// TIA Portal V15.1 export
// export: Created 2022-12-20T09:13:23.4021244Z, ExportSetting None, DisplayName Totally Integrated Automation Portal, DisplayVersion V15.1 Update 1, DisplayName TIA Portal Openness, DisplayVersion V15.1, DisplayName SINAMICS Startdrive Advanced, DisplayVersion V15.1, DisplayName G130, G150, S120, S150, SINAMICS MV, S210, DisplayVersion V15.1, DisplayName G110M, G120, G120C, G120D, G120P, DisplayVersion V15.1, DisplayName STEP 7 Professional, DisplayVersion V15.1 Update 1, DisplayName STEP 7 Safety, DisplayVersion V15.1, DisplayName WinCC Professional, DisplayVersion V15.1 Update 1, DisplayName SIMATIC Visualization Architect, DisplayVersion V15.1
FUNCTION_BLOCK "SA01_MISCELLANEOUS_FB"   // FB905, FBD
TITLE = SA01_MISCELLANEOUS_FB
{ S7_Optimized_Access := 'TRUE' }
// The block is used to control equipment that is not linked to PLC, one SA or one EM
// stored: AutoNumber false, MemoryReserve 100, SetENOAutomatically False
   VAR
      "000-400K18" : "CM_Relay_FB";   // ++000+400-K18
      "000-401K2" : "CM_Relay_FB";   // ++000+401-K2 24VDC Release output station 10
      "000-401K10" : "CM_Relay_FB";   // ++000+401-K10 24VDC Release output station 40
      "000-401K18" : "CM_Relay_FB";   // ++000+401-K18 24VDC Release output station 50
      "000-ZP01-11Y" : "CM_Dump_Valve_FB";   // 000-ZP01-11Y Zone panel dumpvalve
   END_VAR
BEGIN

REGION Network 1: ***Zonepanel***
END_REGION

REGION Network 2: Call relay ++000+400K18
   // 24VDC release zone panel
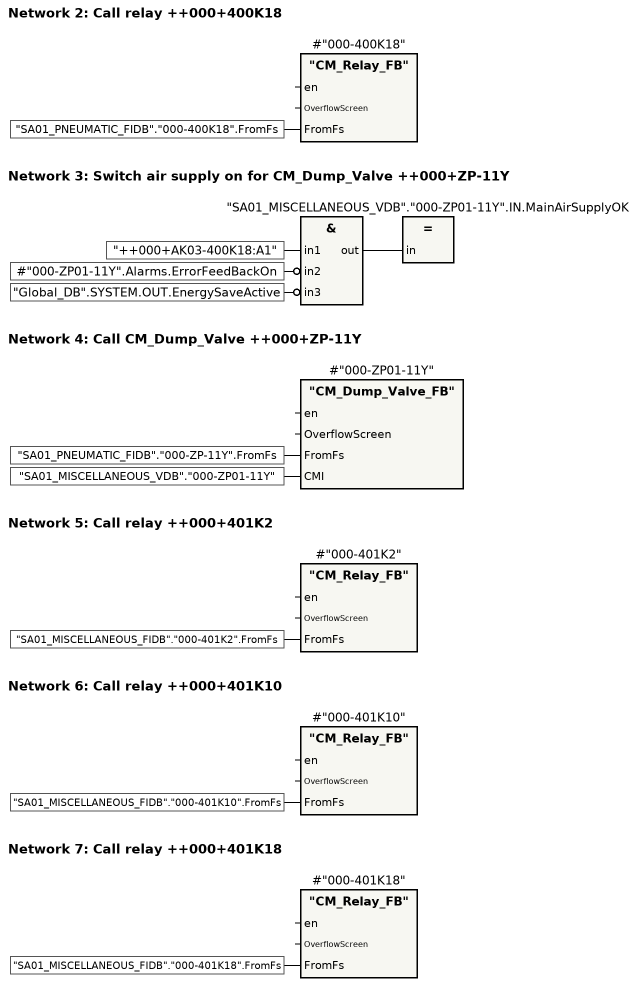
   #"000-400K18"(FromFs := "SA01_PNEUMATIC_FIDB"."000-400K18".FromFs);   // "CM_Relay_FB"
END_REGION

REGION Network 3: Switch air supply on for CM_Dump_Valve ++000+ZP-11Y
   // Set condition to switch air supply on
   "SA01_MISCELLANEOUS_VDB"."000-ZP01-11Y".IN.MainAirSupplyOK := "++000+AK03-400K18:A1" AND NOT #"000-ZP01-11Y".Alarms.ErrorFeedBackOn AND NOT "Global_DB".SYSTEM.OUT.EnergySaveActive;
END_REGION

REGION Network 4: Call CM_Dump_Valve ++000+ZP-11Y
   // Safety function is called SA01_Pneumatic_FBB
   // 000-ZP-11Y always on but switched with the US2 power of the module by a Pilz relay
   #"000-ZP01-11Y"(FromFs := "SA01_PNEUMATIC_FIDB"."000-ZP-11Y".FromFs,   // "CM_Dump_Valve_FB"
                   CMI := "SA01_MISCELLANEOUS_VDB"."000-ZP01-11Y");
END_REGION

REGION Network 5: Call relay ++000+401K2
   // 24VDC Release output station 10
   #"000-401K2"(FromFs := "SA01_MISCELLANEOUS_FIDB"."000-401K2".FromFs);   // "CM_Relay_FB"
END_REGION

REGION Network 6: Call relay ++000+401K10
   // 24VDC Release output station 40
   #"000-401K10"(FromFs := "SA01_MISCELLANEOUS_FIDB"."000-401K10".FromFs);   // "CM_Relay_FB"
END_REGION

REGION Network 7: Call relay ++000+401K18
   // 24VDC Release output station 50
   #"000-401K18"(FromFs := "SA01_MISCELLANEOUS_FIDB"."000-401K18".FromFs);   // "CM_Relay_FB"
END_REGION
END_FUNCTION_BLOCK
